Fanuc KAREL source: kt00060.KL

-- PROVISIONAL review KL for V770-1; original PC SHA256 21f97d1a3bf8289cb1e01ae1c5d0ac36b67c6778303f70ab5bff95bf98a592ce
-- Incomplete behavior may be omitted. Consult companion uncertainty JSON. Do not deploy.
PROGRAM KT00060
%NOLOCKGROUP
VAR
  R2 : REAL
  OUT : REAL
-- UNRESOLVED_DECL H1 type=002017
BEGIN
  -- UNRESOLVED_PC offsets 5-19; opcodes 2E,22,9D,33,B4
  -- UNRESOLVED_PC offsets 24-35; opcodes 2E,23
  -- UNRESOLVED_PC offsets 40-65; opcodes 22,9D,33,B3,21,29,64,29,6A,23
  -- UNRESOLVED_PC offsets 70-74; opcodes 7F
END KT00060
